Omron CX-Programmer project NewProject (CX-Programmer 9.75)

# PLC NewPLC1: CP1L-E EM

## Program NewProgram1 (cyclic task 0)
Local symbols
reset_lamp 100.03 BOOL
start_lamp 100.02 BOOL
start_sw 1.02 BOOL
stop_lamp 100.00 BOOL
stop_sw 1.03 BOOL

### Section Section1

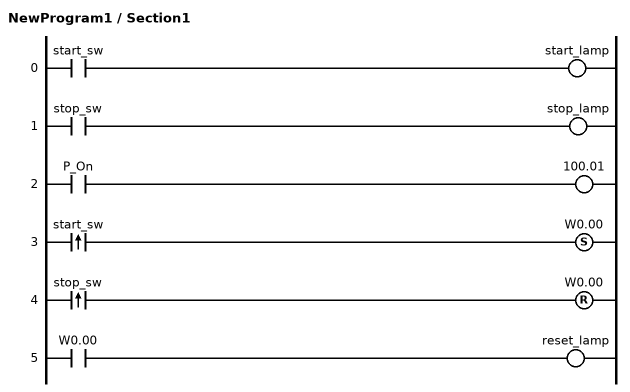
; rung 0
LD start_sw
OUT start_lamp
; rung 1
LD stop_sw
OUT stop_lamp
; rung 2
LD P_On
OUT 100.01
; rung 3
@LD start_sw
SET W0.00
; rung 4
@LD stop_sw
RSET W0.00
; rung 5
LD W0.00
OUT reset_lamp

### Section END
; rung 0
END(001)